PROGRAM UN01_StateMachineRobot_1
VAR
	FB_StateMachineInfeed	: FB_StateManager;
	FB_StateMachinePlacing_1: FB_StateManager;
	FB_StateMachinePlacing_2: FB_StateManager;
	FB_StateMachinePlacing_3: FB_StateManager;
	FB_StateMachinePlacing_4: FB_StateManager;
	FB_StateMachineRobot	: FB_StateManager;
END_VAR

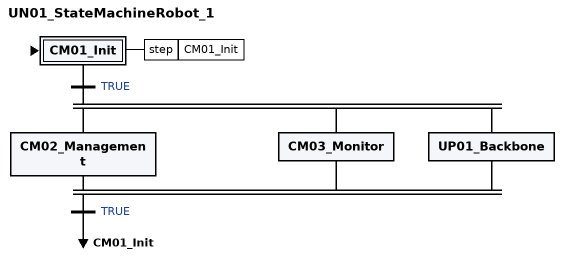
INITIAL_STEP CM01_Init:
    CM01_Init(N);  // step action
END_STEP
TRANSITION FROM CM01_Init TO (CM02_Management, CM03_Monitor, UP01_Backbone)
    := TRUE;
END_TRANSITION
STEP CM02_Management:
END_STEP
STEP CM03_Monitor:
END_STEP
STEP UP01_Backbone:
END_STEP
TRANSITION FROM (CM02_Management, CM03_Monitor, UP01_Backbone) TO CM01_Init
    := TRUE;
END_TRANSITION

ACTION CM01_Init:
//Infeed
Data_GVL.bFL_StartInfeed 			:= Data_GVL.bStartButton OR HMI_GVL.bStartButtonInfeed;
Data_GVL.bFL_StopInfeed 			:= Data_GVL.bStopButton OR HMI_GVL.bStopButtonInfeed;
Data_GVL.bFL_ResetInfeed 			:= Data_GVL.bResetButton OR HMI_GVL.bResetButtonInfeed;
Data_GVL.bFL_AutoManuaModeInfeed 	:= NOT Data_GVL.StateMachineInfeed.Running AND HMI_GVL.bTestModeEnableInfeed;
//Placing 1
Data_GVL.bFL_StartPlacing_1 		:= Data_GVL.bStartButton OR HMI_GVL.bStartButtonPlacing_1;
Data_GVL.bFL_StopPlacing_1 			:= Data_GVL.bStopButton OR HMI_GVL.bStopButtonPlacing_1;
Data_GVL.bFL_ResetPlacing_1			:= Data_GVL.bResetButton OR HMI_GVL.bResetButtonPlacing_1;
Data_GVL.bFL_AutoManuaModePlacing_1 := NOT Data_GVL.StateMachinePlacing_1.Running AND HMI_GVL.bTestModeEnablePlacing_1;
//Placing 2
Data_GVL.bFL_StartPlacing_2 		:= Data_GVL.bStartButton OR HMI_GVL.bStartButtonPlacing_2;
Data_GVL.bFL_StopPlacing_2 			:= Data_GVL.bStopButton OR HMI_GVL.bStopButtonPlacing_2;
Data_GVL.bFL_ResetPlacing_2			:= Data_GVL.bResetButton OR HMI_GVL.bResetButtonPlacing_2;
Data_GVL.bFL_AutoManuaModePlacing_2 := NOT Data_GVL.StateMachinePlacing_2.Running AND HMI_GVL.bTestModeEnablePlacing_2;
//Placing 3
Data_GVL.bFL_StartPlacing_3 		:= Data_GVL.bStartButton OR HMI_GVL.bStartButtonPlacing_3;
Data_GVL.bFL_StopPlacing_3 			:= Data_GVL.bStopButton OR HMI_GVL.bStopButtonPlacing_3;
Data_GVL.bFL_ResetPlacing_3			:= Data_GVL.bResetButton OR HMI_GVL.bResetButtonPlacing_3;
Data_GVL.bFL_AutoManuaModePlacing_3 := NOT Data_GVL.StateMachinePlacing_3.Running AND HMI_GVL.bTestModeEnablePlacing_3;
//Placing 4
Data_GVL.bFL_StartPlacing_4 		:= Data_GVL.bStartButton OR HMI_GVL.bStartButtonPlacing_4;
Data_GVL.bFL_StopPlacing_4 			:= Data_GVL.bStopButton OR HMI_GVL.bStopButtonPlacing_4;
Data_GVL.bFL_ResetPlacing_4			:= Data_GVL.bResetButton OR HMI_GVL.bResetButtonPlacing_4;
Data_GVL.bFL_AutoManuaModePlacing_4 := NOT Data_GVL.StateMachinePlacing_4.Running AND HMI_GVL.bTestModeEnablePlacing_4;
//Robot
Data_GVL.bFL_StartRobot 			:= Data_GVL.bStartButton OR HMI_GVL.bStartButtonRobot;
Data_GVL.bFL_StopRobot 				:= Data_GVL.bStopButton OR HMI_GVL.bStopButtonRobot;
Data_GVL.bFL_ResetRobot 			:= Data_GVL.bResetButton OR HMI_GVL.bResetButtonRobot;
Data_GVL.bFL_AutoManuaModeRobot 	:= NOT Data_GVL.StateMachineRobot.Running AND HMI_GVL.bTestModeEnableRobot;
END_ACTION

ACTION CM02_Management:
// NETWORK 1
END_ACTION

ACTION CM03_Monitor:
// NETWORK 1
END_ACTION

ACTION UP01_Backbone:
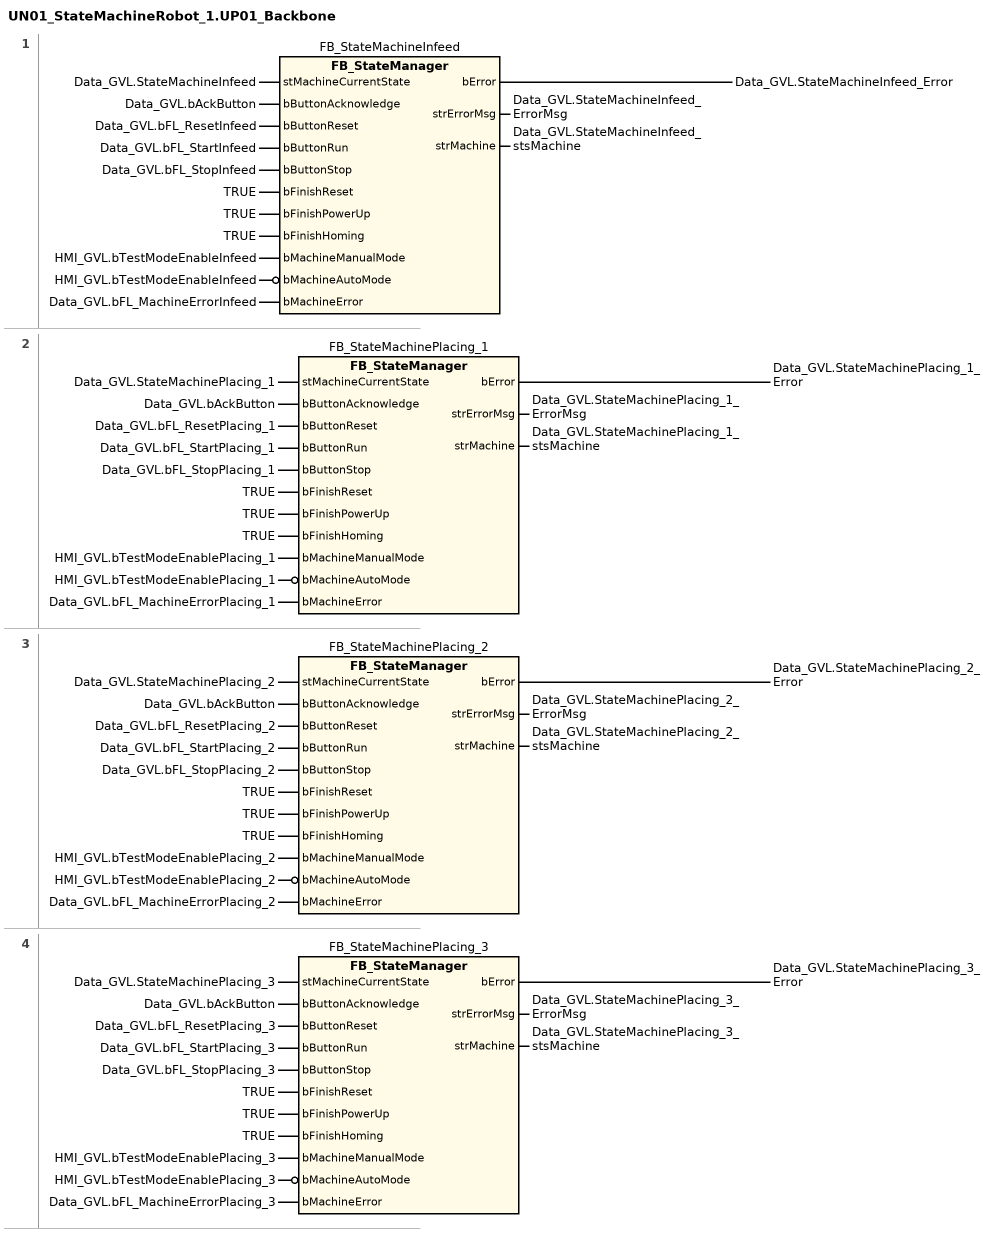
// NETWORK 1
FB_StateMachineInfeed(
    stMachineCurrentState := Data_GVL.StateMachineInfeed,
    bButtonAcknowledge := Data_GVL.bAckButton,
    bButtonReset := Data_GVL.bFL_ResetInfeed,
    bButtonRun := Data_GVL.bFL_StartInfeed,
    bButtonStop := Data_GVL.bFL_StopInfeed,
    bFinishReset := TRUE,
    bFinishPowerUp := TRUE,
    bFinishHoming := TRUE,
    bMachineManualMode := HMI_GVL.bTestModeEnableInfeed,
    bMachineAutoMode := NOT HMI_GVL.bTestModeEnableInfeed,
    bMachineError := Data_GVL.bFL_MachineErrorInfeed,
    strErrorMsg => Data_GVL.StateMachineInfeed_ErrorMsg,
    strMachine => Data_GVL.StateMachineInfeed_stsMachine); // FB_StateManager
Data_GVL.StateMachineInfeed_Error := FB_StateMachineInfeed.bError;

// NETWORK 2
FB_StateMachinePlacing_1(
    stMachineCurrentState := Data_GVL.StateMachinePlacing_1,
    bButtonAcknowledge := Data_GVL.bAckButton,
    bButtonReset := Data_GVL.bFL_ResetPlacing_1,
    bButtonRun := Data_GVL.bFL_StartPlacing_1,
    bButtonStop := Data_GVL.bFL_StopPlacing_1,
    bFinishReset := TRUE,
    bFinishPowerUp := TRUE,
    bFinishHoming := TRUE,
    bMachineManualMode := HMI_GVL.bTestModeEnablePlacing_1,
    bMachineAutoMode := NOT HMI_GVL.bTestModeEnablePlacing_1,
    bMachineError := Data_GVL.bFL_MachineErrorPlacing_1,
    strErrorMsg => Data_GVL.StateMachinePlacing_1_ErrorMsg,
    strMachine => Data_GVL.StateMachinePlacing_1_stsMachine); // FB_StateManager
Data_GVL.StateMachinePlacing_1_Error := FB_StateMachinePlacing_1.bError;

// NETWORK 3
FB_StateMachinePlacing_2(
    stMachineCurrentState := Data_GVL.StateMachinePlacing_2,
    bButtonAcknowledge := Data_GVL.bAckButton,
    bButtonReset := Data_GVL.bFL_ResetPlacing_2,
    bButtonRun := Data_GVL.bFL_StartPlacing_2,
    bButtonStop := Data_GVL.bFL_StopPlacing_2,
    bFinishReset := TRUE,
    bFinishPowerUp := TRUE,
    bFinishHoming := TRUE,
    bMachineManualMode := HMI_GVL.bTestModeEnablePlacing_2,
    bMachineAutoMode := NOT HMI_GVL.bTestModeEnablePlacing_2,
    bMachineError := Data_GVL.bFL_MachineErrorPlacing_2,
    strErrorMsg => Data_GVL.StateMachinePlacing_2_ErrorMsg,
    strMachine => Data_GVL.StateMachinePlacing_2_stsMachine); // FB_StateManager
Data_GVL.StateMachinePlacing_2_Error := FB_StateMachinePlacing_2.bError;

// NETWORK 4
FB_StateMachinePlacing_3(
    stMachineCurrentState := Data_GVL.StateMachinePlacing_3,
    bButtonAcknowledge := Data_GVL.bAckButton,
    bButtonReset := Data_GVL.bFL_ResetPlacing_3,
    bButtonRun := Data_GVL.bFL_StartPlacing_3,
    bButtonStop := Data_GVL.bFL_StopPlacing_3,
    bFinishReset := TRUE,
    bFinishPowerUp := TRUE,
    bFinishHoming := TRUE,
    bMachineManualMode := HMI_GVL.bTestModeEnablePlacing_3,
    bMachineAutoMode := NOT HMI_GVL.bTestModeEnablePlacing_3,
    bMachineError := Data_GVL.bFL_MachineErrorPlacing_3,
    strErrorMsg => Data_GVL.StateMachinePlacing_3_ErrorMsg,
    strMachine => Data_GVL.StateMachinePlacing_3_stsMachine); // FB_StateManager
Data_GVL.StateMachinePlacing_3_Error := FB_StateMachinePlacing_3.bError;

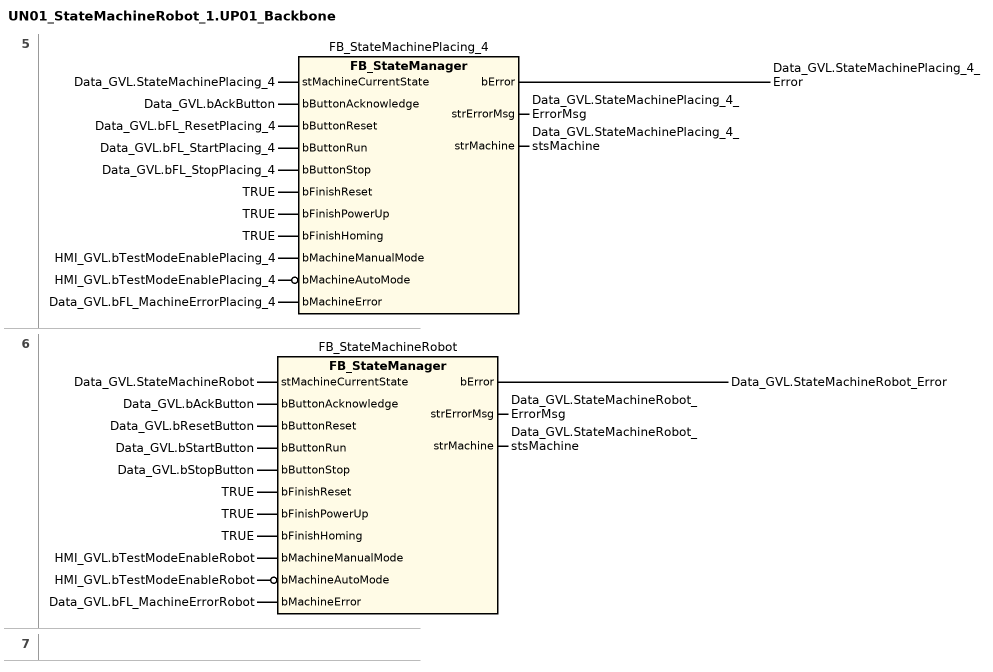
// NETWORK 5
FB_StateMachinePlacing_4(
    stMachineCurrentState := Data_GVL.StateMachinePlacing_4,
    bButtonAcknowledge := Data_GVL.bAckButton,
    bButtonReset := Data_GVL.bFL_ResetPlacing_4,
    bButtonRun := Data_GVL.bFL_StartPlacing_4,
    bButtonStop := Data_GVL.bFL_StopPlacing_4,
    bFinishReset := TRUE,
    bFinishPowerUp := TRUE,
    bFinishHoming := TRUE,
    bMachineManualMode := HMI_GVL.bTestModeEnablePlacing_4,
    bMachineAutoMode := NOT HMI_GVL.bTestModeEnablePlacing_4,
    bMachineError := Data_GVL.bFL_MachineErrorPlacing_4,
    strErrorMsg => Data_GVL.StateMachinePlacing_4_ErrorMsg,
    strMachine => Data_GVL.StateMachinePlacing_4_stsMachine); // FB_StateManager
Data_GVL.StateMachinePlacing_4_Error := FB_StateMachinePlacing_4.bError;

// NETWORK 6
FB_StateMachineRobot(
    stMachineCurrentState := Data_GVL.StateMachineRobot,
    bButtonAcknowledge := Data_GVL.bAckButton,
    bButtonReset := Data_GVL.bResetButton,
    bButtonRun := Data_GVL.bStartButton,
    bButtonStop := Data_GVL.bStopButton,
    bFinishReset := TRUE,
    bFinishPowerUp := TRUE,
    bFinishHoming := TRUE,
    bMachineManualMode := HMI_GVL.bTestModeEnableRobot,
    bMachineAutoMode := NOT HMI_GVL.bTestModeEnableRobot,
    bMachineError := Data_GVL.bFL_MachineErrorRobot,
    strErrorMsg => Data_GVL.StateMachineRobot_ErrorMsg,
    strMachine => Data_GVL.StateMachineRobot_stsMachine); // FB_StateManager
Data_GVL.StateMachineRobot_Error := FB_StateMachineRobot.bError;

// NETWORK 7
END_ACTION

END_PROGRAM

(* stored: Version 1.1.0.1, ProductVersion 3.1.4024.9
   POU UN01_StateMachineRobot_1: Id {95b64d09-2436-46bc-97bc-dc78074d5460}, SpecialFunc None
   Action CM01_Init: Id {d5d18293-afc6-4792-8f3a-9a8fb478cb23}
   Action CM02_Management: Id {c7f37a00-6702-453f-a456-6c8df9ae6a29}
   Action CM03_Monitor: Id {c35c8d73-b022-4f42-977b-80cebb2a733f}
   Action UP01_Backbone: Id {f5710375-27cf-48fe-ae65-38b66efbd6d4} *)
